FUNCTION_BLOCK FB_Pusher
VAR_INPUT
END_VAR
VAR_OUTPUT
	axis_ready				:BOOL:=FALSE;
END_VAR
VAR

PusherServo        			:FB_AxisControl;

_Pusher_param				:recipe;



ToolPositioningSpeed	: LREAL := 20;
ToolPositioningAccel	: LREAL := 100;
ToolPositioningJerk		: LREAL := 1000;
ToolHomingSpeed			: LREAL := 2;

PusherServoEnable			:BOOL;
PusherServoEnabled			:BOOL;

_ExecutedHome				:BOOL:=FALSE;
_ExecutedStage2				:BOOL:=FALSE;
_ExecutedStage4				:BOOL:=FALSE;
_ExecutedStage5				:BOOL:=FALSE;
_ExecutedOffset				:BOOL:=FALSE;
_ExecutedTamp				:BOOL:=FALSE;

tickcounter_pusher: 		INT :=0;
State: 						INT:= 0;
StateNext: 					INT:= 0;

pusher_old_position			:LREAL;




END_VAR

METHOD _absolute_move : BOOL
VAR_INPUT
	Enable				:BOOL;
	Stage				:INT;
END_VAR
IF Enable AND NOT axis_ready THEN
	CASE State OF
	
	0:	
		
		PusherServo.fPosition:= _Pusher_Param.Pusher.Distance[Stage];
		PusherServo.fVelocity:= _Pusher_Param.Pusher.Speed[Stage]; //mm/s
	
		IF stage = 6 THEN
			_Pusher_Param.Clamp.Release_Instance := _Pusher_Param.Clamp.Release_Instance - _Pusher_Param.Pusher.Distance[5];
		
			IF _Pusher_Param.Clamp.Release_Instance <= 0 THEN
				IF qxClamp = TRUE THEN
					qxClamp:=FALSE;
					PRG_Machine.StopClampTimer();
	
				END_IF
			END_IF
	
			pusher_old_position:= PusherServo.fActualPosition;
		END_IF 
		
		PusherServo.xMoveA:=TRUE;
	
	
		StateNext:=5;
	5:	
		IF PusherServo.xInPosition = TRUE THEN
		
			PusherServo.xMoveA := FALSE;
			StateNext:=0;
			axis_ready:=TRUE;
		
			IF qxClamp = TRUE AND Stage = 6 THEN
				qxClamp:=FALSE;
		
				PRG_Machine.StopClampTimer();
	
			END_IF
		END_IF
		
		IF (PusherServo.fActualPosition-pusher_old_position) >= (_Pusher_Param.Clamp.Release_Instance) AND Stage = 6 THEN
			IF qxClamp = TRUE THEN
				qxClamp:=FALSE;
		
				PRG_Machine.StopClampTimer();
	
			END_IF
		END_IF


	END_CASE

	State:=StateNext;
ELSIF NOT enable THEN 
	axis_ready:=FALSE;
	PusherServo.xMoveA := FALSE;
	state:=0;
	statenext:=0;
END_IF
END_METHOD

METHOD _Enable 
VAR_INPUT
END_VAR

PusherServoEnable := TRUE;
END_METHOD

METHOD _force_home  : BOOL
VAR_INPUT
	Enable				:BOOL;
	
END_VAR
IF enable AND NOT axis_ready THEN
	CASE State OF
	
	0:	
	
		PusherServo.fPosition:= 0;
		PusherServo.fVelocity:= 10; //mm/s
	
		PusherServo.xMoveA:=TRUE;
		StateNext:=5;
	5:	
		IF PusherServo.xInPosition = TRUE THEN
		
			PusherServo.xMoveA := FALSE;
			StateNext:=0;
			axis_ready:=TRUE;
		
		END_IF


	END_CASE

	State:=StateNext;
ELSIF NOT enable THEN
	axis_ready:=FALSE;
	PusherServo.xMoveA := FALSE;
	state:=0;
	statenext:=0;
END_IF
END_METHOD

METHOD _Halt : BOOL
VAR_INPUT
END_VAR
PusherServo.xHalt:=TRUE;
END_METHOD

METHOD _Halt_false : BOOL
VAR_INPUT
END_VAR
PusherServo.xHalt:=FALSE;
END_METHOD

METHOD _Home 
VAR_INPUT
	
END_VAR


VAR


END_VAR

VAR_OUTPUT
	
END_VAR


CASE State OF //you are here



0:	
	_ExecutedHome := FALSE;
	PusherServo.fVelocity := ToolPositioningSpeed;
	PusherServo.fAxisAcceleration := ToolPositioningAccel;
	PusherServo.fAxisDeceleration := ToolPositioningAccel;
	PusherServo.fAxisJerk := ToolPositioningJerk;

	IF ixPusherHomeSwitch THEN
		PusherServo.xPositiveDirection := FALSE;
		IF  tickcounter_pusher < 10 THEN
			tickcounter_pusher := tickcounter_pusher + 1;  // can be put in onditional
		
		ELSE
		//IF tickcounter_compress >= 10 THEN
			PusherServo.xMoveV := TRUE;
		END_IF
	ELSE
	
		//CompressServo.xHalt := NOT CompressServo.xHalt;
		PusherServo.xMoveV := FALSE;
		//CompressServo.xHalt := NOT CompressServo.xHalt;
		PusherServo.xHalt := TRUE;
		IF PusherServo.xHalted THEN
			tickcounter_pusher:=0;
			StateNext := 5;
		END_IF
	
	END_IF
	
5:
	
	PusherServo.xHalt := FALSE;
	tickcounter_Pusher := tickcounter_Pusher + 1;
	IF tickcounter_Pusher >= 10 THEN
		tickcounter_Pusher := 0;
		StateNext := 10;
	END_IF
	
10:
	PusherServo.fVelocity := ToolHomingSpeed;
	
	IF NOT ixPusherHomeSwitch THEN
		PusherServo.xPositiveDirection := TRUE;
		IF tickcounter_Pusher < 10 THEN
			tickcounter_Pusher := tickcounter_Pusher + 1;
		ELSE
		//IF tickcounter >= 10 THEN
			PusherServo.xMoveV := TRUE;
		END_IF
	ELSE
		PusherServo.xMoveV := FALSE;
		PusherServo.xHalt := TRUE;
		IF PusherServo.xHalted AND PusherServo.fstandstill THEN
			tickcounter_Pusher := 0;
			StateNext := 15;
		END_IF
	END_IF

15:
	
	PusherServo.xHalt := FALSE;
	tickcounter_Pusher := tickcounter_Pusher + 1;
	IF tickcounter_Pusher >= 25 THEN
		tickcounter_Pusher := 0;
		StateNext := 20;
		//Executed := TRUE;
	END_IF
20:
	PusherServo.fHomeOffset := 0;
	PusherServo.xZero := TRUE;
	StateNext := 25;	
	
25:
	IF PusherServo.xZeroed THEN
		PusherServo.xZero := FALSE;
		_ExecutedHome := TRUE;
		StateNext := 0;
	END_IF
	

END_CASE

State := StateNext;
END_METHOD

METHOD _mc_stop : BOOL
VAR_INPUT
END_VAR
PusherServo.xStop:=TRUE;
END_METHOD

METHOD _Reset
VAR_INPUT
END_VAR
	tickcounter_Pusher:=0;
	PusherServoEnable := FALSE;
	PusherServo.xZero := FALSE;
	PusherServo.xMoveV := FALSE;
	PusherServo.xMoveA := FALSE;
	PusherServo.xHalt := FALSE;
	PusherServo.GearIn := FALSE;
	PusherServo.xStop:=FALSE;
	state:=0;
	statenext:=0;
	
	
	axis_ready:=FALSE;
	_ExecutedHome:=FALSE;
	_ExecutedOffset:=FALSE;
	PRG_Machine.reset_rec_old();
	PRG_Machine._debug(enable:=FALSE);
END_METHOD

METHOD _Reset_medium
VAR_INPUT
END_VAR
	tickcounter_Pusher:=0;
	PusherServoEnable := FALSE;
	PusherServo.xZero := FALSE;
	PusherServo.xMoveV := FALSE;
	PusherServo.xMoveA := FALSE;
	PusherServo.xHalt := FALSE;
	PusherServo.GearIn := FALSE;
	PusherServo.xStop:=FALSE;
	state:=0;
	statenext:=0;
	
	
	axis_ready:=FALSE;
	PRG_Machine._debug(enable:=FALSE);
END_METHOD

METHOD _retract  : BOOL
VAR_INPUT
	Enable				:BOOL;
	
END_VAR
IF enable AND NOT axis_ready THEN
	CASE State OF
	
	0:	
	
		PusherServo.fPosition:= 0;
		PusherServo.fVelocity:= _Pusher_Param.Pusher.Retract_Speed; //mm/s
	
		PusherServo.xMoveA:=TRUE;
		StateNext:=5;
	5:	
		IF PusherServo.xInPosition = TRUE THEN
		
			PusherServo.xMoveA := FALSE;
			StateNext:=0;
			axis_ready:=TRUE;
		
		END_IF


	END_CASE

	State:=StateNext;
ELSIF NOT enable THEN
	axis_ready:=FALSE;
	PusherServo.xMoveA := FALSE;
	state:=0;
	
END_IF
END_METHOD

METHOD _Soft_Reset
VAR_INPUT
END_VAR

tickcounter_Pusher:=0;
PusherServo.xZero := FALSE;
PusherServo.xMoveV := FALSE;
PusherServo.xMoveA := FALSE;
PusherServo.xHalt := FALSE;
PusherServo.GearIn := FALSE;
PusherServo.xStop:=FALSE;
state:=0;
statenext:=0;

axis_ready:=FALSE;
PRG_Machine._debug(enable:=FALSE);
END_METHOD

METHOD _Update
VAR_INPUT
END_VAR
PusherServo(
	xEnable:= PusherServoEnable, 
	xZero:= , 
	xMoveR:= , 
	xMoveA:= , 
	xMoveV:= , 
	xPositiveDirection:= , 
	fDistance:= , 
	fPosition:= , 
	fVelocity:= , 
	xStop:= , 
	xHome:= , 
	xHomeFlag:= , 
	homePosition:=0,
	fActualPosition=> , 
	fActualVelocity=> , 
	fActModuloPos=> , 
	xEnabled=> PusherServoEnabled, 
	xMoveComplete=> , 
	xInPosition=> , 
	xAtSpeed=> , 
	xStopped=> , 
	xHomed=> ,
	errorID=> PusherServoErrorID, 
	Axis:= PusherAxis );
END_METHOD

PROPERTY HomeExecuted : BOOL
GET
HomeExecuted := _ExecutedHome;
END_GET
SET
_ExecutedHome := HomeExecuted;
END_SET
END_PROPERTY

METHOD Offset
VAR_INPUT
	Enable				:BOOL;
END_VAR

IF enable AND NOT axis_ready THEN	
	CASE State OF
	0:	
		_ExecutedOffset:=FALSE;
		PusherServo.fPosition:= _Pusher_Param.Other.Pusher_Home_Offset-PRG_Machine.rec_old.other.pusher_home_offset;
		PusherServo.fVelocity:= 20; //mm/s
	
		IF PusherServo.fPosition<>0 THEN
			PusherServo.xMoveA:=TRUE;
			StateNext:=5;
		ELSE
			_ExecutedOffset:=TRUE;
		END_IF
	
		//StateNext:=5;
	5:	
		IF PusherServo.xInPosition = TRUE AND PusherServo.fstandstill THEN
			
			PusherServo.xMoveA := FALSE;
			StateNext:=7;
			//_ExecutedOffset:=TRUE;
		
		END_IF
	7:
		tickcounter_pusher:=tickcounter_pusher+1;
		IF tickcounter_Pusher >= 25 THEN
			tickcounter_Pusher := 0;
			StateNext := 10;
			//Executed := TRUE;
		END_IF	
	
	10:
	
		PusherServo.fHomeOffset := 0;
		pusherServo.xZero := TRUE;
		StateNext := 15;	
	
	15:
		IF pusherServo.xZeroed THEN
			pusherServo.xZero := FALSE;
			_ExecutedOffset:=TRUE;
			axis_ready:=TRUE;
			StateNext := 0;
		END_IF

	END_CASE

	State:=StateNext;
	
ELSIF NOT enable THEN 
	axis_ready:=FALSE;
	pusherServo.xZero := FALSE;
	StateNext := 0;
END_IF
END_METHOD

PROPERTY OffsetExecuted : BOOL
GET
OffsetExecuted := _ExecutedOffset;
END_GET
SET
_ExecutedOffset := OffsetExecuted;
END_SET
END_PROPERTY

PROPERTY Pusher_Param : recipe
GET
Pusher_param := _Pusher_Param;
END_GET
SET
_Pusher_param := Pusher_Param;
END_SET
END_PROPERTY

PROPERTY Stage2Executed : BOOL
GET
Stage2Executed := _ExecutedStage2;
END_GET
SET
_ExecutedStage2 := Stage2Executed;
END_SET
END_PROPERTY

PROPERTY Stage4Executed : BOOL
GET
Stage4Executed := _ExecutedStage4;
END_GET
SET
_ExecutedStage4 := Stage4Executed;
END_SET
END_PROPERTY

PROPERTY Stage5Executed : BOOL
GET
Stage5Executed := _ExecutedStage5;
END_GET
SET
_ExecutedStage5 := Stage5Executed;
END_SET
END_PROPERTY

PROPERTY TampExecuted : BOOL
GET
TampExecuted := _ExecutedTamp;
END_GET
SET
_ExecutedTamp := TampExecuted;
END_SET
END_PROPERTY

END_FUNCTION_BLOCK

(* stored: Version 1.1.0.1, ProductVersion 3.1.4020.12
   POU FB_Pusher: Id {36e33e78-1ebc-4d07-bdf3-4dd4d01880b2}, SpecialFunc None
   Folder Executed: Id {7a10ea65-564e-4af0-9fe0-b64a71cccc00}
   Folder param: Id {78515c04-73b4-4e21-a577-974d1bbadc16}
   Method _absolute_move: Id {f90b17c3-164d-4ba6-9e40-6e0ce82312ff}
   Method _Enable: Id {6bb019dc-8171-4b90-aa60-df783a0d8ed1}
   Method _force_home: Id {296c7470-8d9d-4d7c-88ab-fbecc02976bb}
   Method _Halt: Id {6dffbb07-095b-46ed-992a-d66a25d3d5b1}
   Method _Halt_false: Id {dc9dee2e-fbf9-425f-97da-465ec9996c5c}
   Method _Home: Id {6f7955b9-e0ab-4bc1-b9ef-99b4a74065aa}
   Method _mc_stop: Id {7e9e7bd5-2c2f-4617-90fa-1a4a9040aed4}
   Method _Reset: Id {13afff2a-b85d-41c3-909c-3571ef832fac}
   Method _Reset_medium: Id {d0af1c72-badd-4f28-b191-8a590c1ea4f5}
   Method _retract: Id {a4ed0cb5-2786-4aab-b82d-9d2e31076ef4}
   Method _Soft_Reset: Id {6dfb29ba-6c3e-40e5-9d3b-23a15f2e4bb6}
   Method _Update: Id {c072dfad-6af6-4653-b890-372b04534df9}
   Property HomeExecuted: Id {c4909d4e-7cc6-4c8a-a82b-5891d80aff66}
   Get Get: Id {777dec52-37c9-4f1c-95e1-158ef6c4608a}
   Set Set: Id {3302950f-7a49-4729-923a-16e7c9debbf0}
   Method Offset: Id {26b497cf-7aad-4dd1-9640-d61454ccb044}
   Property OffsetExecuted: Id {008d4b7a-397f-4e6a-89a4-4ea230bddc80}
   Get Get: Id {7199c352-dbae-48f9-ba6f-85d625beb146}
   Set Set: Id {ce6c7ecb-29b5-49a1-b805-b11f3e4bfc24}
   Property Pusher_Param: Id {6122f36e-b405-439e-9b5e-88ea35c81274}
   Get Get: Id {4560b3aa-fa7b-487d-929f-959b9a24e9ca}
   Set Set: Id {669869ab-c4ac-483b-a636-e778db41462a}
   Property Stage2Executed: Id {f3289000-cd18-410c-b583-9cf1ce52a86d}
   Get Get: Id {e6259f44-f305-4fbc-980e-4a546b857acd}
   Set Set: Id {6653e3b4-31ed-433a-b44b-2b6b0932413c}
   Property Stage4Executed: Id {936c5c19-dc5f-4e08-a2fb-6dceba308d0a}
   Get Get: Id {bd1e5a73-304d-4a37-9a10-215241e8b902}
   Set Set: Id {5fc62e27-39c6-45f8-9f0b-96a190a876dc}
   Property Stage5Executed: Id {a1eb5161-5bff-4b17-87fa-374af998095e}
   Get Get: Id {2a31c805-c50a-4d2c-9f85-38339fe591e8}
   Set Set: Id {947fcb3d-3774-4aac-b373-d3e03a0a6d4e}
   Property TampExecuted: Id {1ce40493-7a02-4274-b1ae-bfa4312519da}
   Get Get: Id {e2d4d081-fd02-496c-84ae-7dad4bc0c8ee}
   Set Set: Id {04c8e692-b6dc-4358-9473-827608e7f7f1} *)
